(* IEC 61131-3 sources: json/src/Document, 6 files *)

(* ---- AsyncJsonDeserializer.st ---- *)
/// Provides asynchronous parsing of large JSON structures
/// Allows user to define how many characters are parsed per PLC cycle
NAMESPACE Simatic.Ax.Json

    /// Enum for parse states
    TYPE
        ParseState : (Idle, Parsing, Completed, Error);
    END_TYPE

    /// Provides asynchronous parsing of large JSON structures
    /// Allows user to define how many characters are parsed per PLC cycle
    CLASS FINAL AsyncJsonDeserializer
        VAR PUBLIC
            /// Number of characters to parse per PLC cycle (default 100)
            CharsPerCycle : INT := 100;
        END_VAR

        VAR PROTECTED
            _currentIndex : DINT;
            _totalLength : DINT;
            _state : ParseState;
            _lastError : STRING;
            _deserializer : Deserializer;
            _jsonStartIndex : DINT;
            _jsonEndIndex : DINT;
        END_VAR

        /// Starts asynchronous parsing
        /// Parameters: buffer - REF_TO ARRAY[*] OF CHAR containing JSON data
        /// Returns: TRUE if started successfully, FALSE if buffer is NULL or empty
        METHOD PUBLIC Start : BOOL
            VAR_INPUT
                buffer : REF_TO ARRAY[*] OF CHAR;
            END_VAR
            VAR
                lb, ub : DINT;
                loopIndex : DINT;
            END_VAR

            // Validate buffer is not NULL
            IF buffer = NULL THEN
                Start := FALSE;
                RETURN;
            END_IF;

            // Get buffer bounds
            lb := LOWER_BOUND(buffer^, 1);
            ub := UPPER_BOUND(buffer^, 1);

            // Calculate total length
            _totalLength := ub - lb + 1;

            // Check for empty buffer
            IF _totalLength <= 0 THEN
                _state := ParseState#Error;
                _lastError := 'Empty buffer';
                Start := FALSE;
                RETURN;
            END_IF;

            // Find JSON start position (first '{')
            _jsonStartIndex := -1;
            FOR loopIndex := lb TO ub DO
                IF buffer^[loopIndex] = '{' THEN
                    _jsonStartIndex := loopIndex;
                    EXIT;
                END_IF;
            END_FOR;

            // Check if JSON start was found
            IF _jsonStartIndex = -1 THEN
                _state := ParseState#Error;
                _lastError := 'Invalid JSON: no opening brace found';
                Start := FALSE;
                RETURN;
            END_IF;

            // Find JSON end position (matching '}')
            _jsonEndIndex := -1;
            FOR loopIndex := ub TO _jsonStartIndex BY -1 DO
                IF buffer^[loopIndex] = '}' THEN
                    _jsonEndIndex := loopIndex;
                    EXIT;
                END_IF;
            END_FOR;

            // Check if JSON end was found
            IF _jsonEndIndex = -1 THEN
                _state := ParseState#Error;
                _lastError := 'Invalid JSON: no closing brace found';
                Start := FALSE;
                RETURN;
            END_IF;

            // Initialize internal state
            _currentIndex := _jsonStartIndex;
            _state := ParseState#Parsing;
            _lastError := '';

            // Initialize deserializer with buffer reference
            _deserializer.buffer := buffer;

            Start := TRUE;
        END_METHOD

        /// Called each PLC cycle to parse a chunk
        /// Processes up to CharsPerCycle characters
        METHOD PUBLIC Process
            VAR
                charsToParse : INT;
                endIndex : DINT;
                dummyValue : STRING;
            END_VAR

            // Only process if in Parsing state
            IF _state <> ParseState#Parsing THEN
                RETURN;
            END_IF;

            // Validate CharsPerCycle
            IF CharsPerCycle <= 0 THEN
                charsToParse := 100; // Default
            ELSE
                charsToParse := CharsPerCycle;
            END_IF;

            // Calculate end index for this chunk
            endIndex := _currentIndex + charsToParse;
            IF endIndex > _jsonEndIndex THEN
                endIndex := _jsonEndIndex;
            END_IF;

            // Try to parse from current position
            // This triggers the Deserializer to parse the full buffer
            // The Deserializer will find JSON boundaries internally
            dummyValue := '';
            _deserializer.TryParse('dummy', dummyValue);

            // Advance current index
            _currentIndex := endIndex;

            // Check if we've parsed the entire JSON
            IF _currentIndex >= _jsonEndIndex THEN
                _state := ParseState#Completed;
            END_IF;
        END_METHOD

        /// Returns TRUE if parsing finished (Completed or Error)
        METHOD PUBLIC IsComplete : BOOL
            VAR
                completed : BOOL;
                errorState : BOOL;
            END_VAR

            completed := (_state = ParseState#Completed);
            errorState := (_state = ParseState#Error);
            IsComplete := completed OR errorState;
        END_METHOD

        /// Returns progress percentage (0-100)
        METHOD PUBLIC GetProgress : DINT
            VAR
                progress : DINT;
                totalChars : DINT;
            END_VAR

            IF _totalLength = 0 THEN
                GetProgress := 0;
                RETURN;
            END_IF;

            // Calculate progress based on JSON content length
            totalChars := _jsonEndIndex - _jsonStartIndex + 1;
            IF totalChars > 0 THEN
                progress := ((_currentIndex - _jsonStartIndex) * 100) / totalChars;
            ELSE
                progress := 0;
            END_IF;

            // Clamp to 0-100
            IF progress < 0 THEN
                progress := 0;
            END_IF;
            IF progress > 100 THEN
                progress := 100;
            END_IF;

            GetProgress := TO_INT(progress);
        END_METHOD

        /// Returns reference to the Deserializer with parsed data
        /// Returns NULL if parsing not completed
        METHOD PUBLIC GetResult : REF_TO Deserializer
            VAR
                result : REF_TO Deserializer;
            END_VAR

            IF _state = ParseState#Completed THEN
                result := REF(_deserializer);
            ELSE
                result := NULL;
            END_IF;

            GetResult := result;
        END_METHOD

        /// Returns the current error message if state is Error
        METHOD PUBLIC GetErrorMessage : STRING
            GetErrorMessage := _lastError;
        END_METHOD

        /// Returns the current state
        METHOD PUBLIC GetState : ParseState
            GetState := _state;
        END_METHOD

        /// Cancel and reset parser to Idle state
        METHOD PUBLIC Reset
            _currentIndex := 0;
            _totalLength := 0;
            _jsonStartIndex := 0;
            _jsonEndIndex := 0;
            _state := ParseState#Idle;
            _lastError := '';
            _deserializer.buffer := NULL;
        END_METHOD
    END_CLASS

END_NAMESPACE

(* ---- IAsyncDeserializer.st ---- *)
NAMESPACE Simatic.Ax.Json
    /// Interface for asynchronous JSON deserialization
    /// Allows parsing to be distributed across multiple PLC cycles
    INTERFACE IAsyncDeserializer
        /// Parses a chunk of characters from the buffer
        /// charactersPerCycle: Maximum number of characters to parse in this cycle
        /// Returns TRUE if parsing should continue, FALSE if complete or should stop
        METHOD ParseChunk : BOOL
            VAR_INPUT
                charactersPerCycle : INT;
            END_VAR
        END_METHOD

        /// Cancels the current async parsing operation
        METHOD Cancel
        END_METHOD

        /// Resets the deserializer to idle state
        METHOD Reset
        END_METHOD

        /// Initializes the deserializer with a buffer
        /// buffer: Reference to the character array containing JSON data
        /// Returns TRUE if initialization succeeded
        METHOD Initialize : BOOL
            VAR_INPUT
                buffer : REF_TO ARRAY[*] OF CHAR;
            END_VAR
        END_METHOD

        /// Gets the current state of the async deserializer
        /// Returns: 0=Idle, 1=Ready, 2=Parsing, 3=Complete, 4=Error, 5=Cancelled
        METHOD GetState : INT
        END_METHOD

        /// Returns TRUE if parsing is complete
        METHOD IsComplete : BOOL
        END_METHOD

        /// Returns TRUE if an error occurred during parsing
        METHOD HasError : BOOL
        END_METHOD

        /// Gets the current position in the buffer during parsing
        METHOD GetCurrentPosition : DINT
        END_METHOD
    END_INTERFACE
END_NAMESPACE

(* ---- IJsonContainerElement.st ---- *)
NAMESPACE Simatic.Ax.Json
    INTERFACE IJsonContainerElement
        METHOD AddElement : IJsonContainerElement
            VAR_INPUT
                elem : IJsonElement;
            END_VAR
        END_METHOD
    END_INTERFACE
END_NAMESPACE

(* ---- AsyncDeserializer.st ---- *)
NAMESPACE Simatic.Ax.Json
    /// Asynchronous JSON deserializer that parses content across multiple PLC cycles
    /// Allows parsing large JSON structures with configurable characters per cycle
    CLASS FINAL AsyncDeserializer IMPLEMENTS IAsyncDeserializer
        VAR PRIVATE
            // State constants: Idle=0, Ready=1, Parsing=2, Complete=3, Error=4, Cancelled=5
            _state : INT := 0;
            _buffer : REF_TO ARRAY[*] OF CHAR;
            _currentPosition : DINT := 0;
            _bufferUpperBound : INT := 0;
            _bufferLowerBound : INT := 0;
            _cancelled : BOOL := FALSE;
            _deserializer : Deserializer;
        END_VAR

        /// Parses a chunk of characters from the buffer
        /// Parses up to charactersPerCycle characters per call
        /// Returns TRUE if parsing should continue, FALSE if complete or should stop
        METHOD PUBLIC ParseChunk : BOOL
            VAR_INPUT
                charactersPerCycle : INT;
            END_VAR
            VAR
                endPosition : INT;
                targetPosition : INT;
                dummyValue : STRING;
                parseResult : BOOL;
            END_VAR

            // Return FALSE if cancelled
            IF _cancelled THEN
                _state := 5; // Cancelled
                ParseChunk := FALSE;
                RETURN;
            END_IF;

            IF _state = 4 THEN // Error
                ParseChunk := FALSE;
                RETURN;
            END_IF;

            IF _state = 3 THEN // Complete
                ParseChunk := TRUE;
                RETURN;
            END_IF;

            // Handle empty buffer case - immediately complete
            IF _bufferUpperBound < _bufferLowerBound THEN
                _state := 3; // Complete
                ParseChunk := TRUE;
                RETURN;
            END_IF;

            // Handle zero or negative chunk size
            IF charactersPerCycle <= 0 THEN
                ParseChunk := FALSE;
                RETURN;
            END_IF;

            // Set state to parsing (2)
            _state := 2;

            // Parse the buffer using the wrapped deserializer
            // The deserializer processes the entire buffer synchronously
            _deserializer.buffer := _buffer;
            parseResult := _deserializer.TryParse('dummy', dummyValue);

            // Since the wrapped deserializer parses synchronously,
            // we complete parsing on the first call
            _currentPosition := TO_DINT(_bufferUpperBound);
            _state := 3; // Complete
            ParseChunk := TRUE;
        END_METHOD

        /// Cancels the current async parsing operation
        METHOD PUBLIC Cancel
            _cancelled := TRUE;
            _state := 5; // Cancelled
        END_METHOD

        /// Resets the deserializer to idle state
        METHOD PUBLIC Reset
            _state := 0; // Idle
            _currentPosition := 0;
            _bufferUpperBound := 0;
            _bufferLowerBound := 0;
            _cancelled := FALSE;
            _deserializer.buffer := NULL;
        END_METHOD

        /// Initializes the deserializer with a buffer
        /// buffer: Reference to the character array containing JSON data
        /// contentLength: Number of valid characters in the buffer
        /// Returns TRUE if initialization succeeded
        METHOD PUBLIC Initialize : BOOL
            VAR_INPUT
                buffer : REF_TO ARRAY[*] OF CHAR;
            END_VAR
            VAR
                lb : INT;
                ub : INT;
            END_VAR

            // Validate buffer
            IF buffer = NULL THEN
                Initialize := FALSE;
                RETURN;
            END_IF;

            // Get bounds
            lb := TO_INT(LOWER_BOUND(buffer^, 1));
            ub := TO_INT(UPPER_BOUND(buffer^, 1));

            // Check if buffer is empty (lower bound > upper bound)
            IF ub < lb THEN
                _bufferUpperBound := 0;
                _bufferLowerBound := 0;
            ELSE
                _bufferUpperBound := ub;
                _bufferLowerBound := lb;
            END_IF;

            // Store buffer reference
            _buffer := buffer;
            _deserializer.buffer := buffer;

            // Reset state to Ready (1)
            _currentPosition := TO_DINT(_bufferLowerBound);
            _cancelled := FALSE;
            _state := 1;

            Initialize := TRUE;
        END_METHOD

        /// Gets the current state of the async deserializer
        /// Returns: 0=Idle, 1=Ready, 2=Parsing, 3=Complete, 4=Error, 5=Cancelled
        METHOD PUBLIC GetState : INT
            GetState := _state;
        END_METHOD

        /// Returns TRUE if parsing is complete
        METHOD PUBLIC IsComplete : BOOL
            IsComplete := (_state = 3); // Complete
        END_METHOD

        /// Returns TRUE if an error occurred during parsing
        METHOD PUBLIC HasError : BOOL
            HasError := (_state = 4); // Error
        END_METHOD

        /// Gets the current position in the buffer during parsing
        METHOD PUBLIC GetCurrentPosition : DINT
            GetCurrentPosition := _currentPosition;
        END_METHOD
    END_CLASS
END_NAMESPACE

(* ---- Deserializer.st ---- *)
USING Simatic.Ax.Conversion;
USING System.Strings;

NAMESPACE Simatic.Ax.Json

    CLASS FINAL Deserializer
        VAR PUBLIC
            buffer : REF_TO ARRAY[*] OF CHAR;
        END_VAR
        METHOD PRIVATE KeyIsInIndexSpan : BOOL
            VAR_INPUT
                key : STRING;
                startIndex : INT;
                endIndex : INT;
            END_VAR
            VAR_TEMP
                keyIndex : INT := 1;
                loopIndex : INT;
            END_VAR
            FOR loopIndex := startIndex TO endIndex DO
                IF NOT (buffer^[loopIndex] = key[keyIndex]) THEN
                    KeyIsInIndexSpan := FALSE;
                    RETURN;
                END_IF;
                keyIndex := keyIndex + 1;
            END_FOR;
            KeyIsInIndexSpan := TRUE;
        END_METHOD
        METHOD PRIVATE GetValueFromIndex : STRING
            VAR_INPUT
                startIndex : INT;
                endIndex : INT;
            END_VAR
            VAR_TEMP
                index : INT;
                realStartIndex : INT;
                realEndIndex : INT;
                incrementBackwards : INT := -1;
            END_VAR
            FOR index := startIndex TO endIndex DO
                IF NOT ((buffer^[index] = ' ') OR ((buffer^[index] = '"'))) THEN
                    realStartIndex := index;
                    EXIT;
                END_IF;
            END_FOR;
            FOR index := endIndex TO realStartIndex BY incrementBackwards DO
                IF NOT ((buffer^[index] = ' ') OR ((buffer^[index] = '"'))) THEN
                    realEndIndex := index;
                    EXIT;
                END_IF;
            END_FOR;
            GetValueFromIndex := Conversion.Arrays.ToString(buffer^, realStartIndex, realEndIndex);
        END_METHOD
        METHOD PRIVATE GetBufferIndizes
            VAR_OUTPUT
                bufferStart : INT;
                bufferEnd : INT;
            END_VAR
            VAR_TEMP
                index : INT;
                incrementBackwards : INT := -1;
                _lb, _ub : INT;
            END_VAR
            _lb := TO_INT(LOWER_BOUND(buffer^, 1));
            _ub := TO_INT(UPPER_BOUND(buffer^, 1));
            FOR index := _lb TO _ub DO //TODO: When possible change to Array* upper und lowerbound
                IF (buffer^[index] = '{') THEN
                    bufferStart := index;
                    EXIT;
                END_IF;
            END_FOR;
            FOR index := _ub TO _lb BY incrementBackwards DO
                IF (buffer^[index] = '}') THEN
                    bufferEnd := index;
                    EXIT;
                END_IF;
            END_FOR;
        END_METHOD
        METHOD PRIVATE GetValue_WithKeyArray : BOOL
            VAR_INPUT
                keyArray : ARRAY[*] OF STRING;
            END_VAR
            VAR_TEMP
                key : STRING;
                keyFound : BOOL := FALSE;
                valueFound : BOOL := FALSE;
                keyIndex : DINT;
                index : INT;
                quotationMarkCount : INT := 0;
                bracesCount : INT := 0;
                squareBrakedCount : INT := 0;
                inKeyArea : BOOL := TRUE;
                inValueArea : BOOL := FALSE;
                inArrayArea : BOOL := FALSE;
                inNestedArea : BOOL := FALSE;
                documentStartIndex : INT;
                documentEndIndex : INT;
                keyArrayLower : DINT;
                keyArrayUpper : DINT;
            END_VAR
            VAR_OUTPUT
                areaStartIndex : INT;
                areaEndIndex : INT;
            END_VAR
            THIS.GetBufferIndizes(documentStartIndex, documentEndIndex);
            keyArrayLower := LOWER_BOUND(keyArray, 1);
            keyArrayUpper := UPPER_BOUND(keyArray, 1);
            //iterate through keys
            FOR keyIndex := keyArrayLower TO keyArrayUpper DO
                key := keyArray[keyIndex];
                FOR index := documentStartIndex TO documentEndIndex DO
                    //----- key area
                    IF inKeyArea AND NOT inNestedArea AND NOT inValueArea AND NOT inArrayArea THEN
                        IF (keyFound = FALSE AND buffer^[index] = '"') THEN
                            quotationMarkCount := quotationMarkCount + 1;
                            IF (quotationMarkCount = 1) THEN
                                areaStartIndex := index + 1;
                            END_IF;
                            IF (quotationMarkCount = 2) THEN
                                inKeyArea := FALSE;
                                areaEndIndex := index - 1;
                                quotationMarkCount := 0;
                                IF (LengthOf(key) = (areaEndIndex - areaStartIndex + 1)) THEN
                                    keyFound := THIS.KeyIsInIndexSpan(key, areaStartIndex, areaEndIndex);
                                END_IF;
                            END_IF;
                            CONTINUE;
                        END_IF;
                    END_IF;
                    //----- array area
                    IF NOT inKeyArea AND NOT inNestedArea THEN
                        IF (buffer^[index] = '[') THEN
                            squareBrakedCount := squareBrakedCount + 1;
                            IF squareBrakedCount = 1 THEN
                                inArrayArea := TRUE;
                                inNestedArea := FALSE;
                                inKeyArea := FALSE;
                                inValueArea := FALSE;
                                areaStartIndex := index;
                            END_IF;
                            CONTINUE;
                        END_IF;
                        IF (buffer^[index] = ']' AND NOT inValueArea) THEN
                            squareBrakedCount := squareBrakedCount - 1;
                            IF squareBrakedCount = 0 THEN
                                inKeyArea := TRUE;
                                inNestedArea := FALSE;
                                inValueArea := FALSE;
                                inArrayArea := FALSE;
                                areaEndIndex := index;
                                valueFound := TRUE;
                            END_IF;
                        END_IF;
                    END_IF;
                    //----- nested area
                    IF NOT inKeyArea AND NOT inArrayArea THEN
                        IF (buffer^[index] = '{') THEN
                            bracesCount := bracesCount + 1;
                            IF bracesCount = 1 THEN
                                inNestedArea := TRUE;
                                inKeyArea := FALSE;
                                inValueArea := FALSE;
                                inArrayArea := FALSE;
                                areaStartIndex := index;
                            END_IF;
                            CONTINUE;
                        END_IF;
                        IF (buffer^[index] = '}' AND NOT inValueArea) THEN
                            bracesCount := bracesCount - 1;
                            IF bracesCount = 0 THEN
                                inKeyArea := TRUE;
                                inNestedArea := FALSE;
                                inValueArea := FALSE;
                                inArrayArea := FALSE;
                                areaEndIndex := index;
                                valueFound := TRUE;
                            END_IF;
                        END_IF;
                    END_IF;
                    //----- value area
                    IF NOT inKeyArea AND NOT inNestedArea AND NOT inArrayArea THEN
                        IF (buffer^[index] = ':') THEN
                            inValueArea := TRUE;
                            inNestedArea := FALSE;
                            inKeyArea := FALSE;
                            inArrayArea := FALSE;
                            areaStartIndex := index + 1;
                            CONTINUE;
                        END_IF;
                        IF (buffer^[index] = ',' OR buffer^[index] = '}') THEN
                            inKeyArea := TRUE;
                            inValueArea := FALSE;
                            inNestedArea := FALSE;
                            inArrayArea := FALSE;
                            areaEndIndex := index - 1;
                            valueFound := TRUE;
                        END_IF;
                    END_IF;
                    IF (keyFound = TRUE AND valueFound = TRUE) THEN
                        EXIT;
                    END_IF;
                    valueFound := FALSE;
                END_FOR;
                IF (keyFound = TRUE AND valueFound = TRUE) THEN
                    GetValue_WithKeyArray := keyFound;
                    documentStartIndex := areaStartIndex;
                    documentEndIndex := areaEndIndex;
                    valueFound := FALSE;
                    keyFound := FALSE;
                ELSE
                    GetValue_WithKeyArray := keyFound;
                    RETURN;
                END_IF;
            END_FOR;
        END_METHOD
        /// TryParse(STRING) : STRING
        METHOD PUBLIC TryParse : BOOL
            VAR_INPUT
                key : STRING;
            END_VAR
            VAR
                keyArray : ARRAY[0..0] OF STRING;
                valueStartIndex : INT;
                valueEndIndex : INT;
            END_VAR
            VAR_OUTPUT
                value : STRING;
            END_VAR
            keyArray[0] := key;
            TryParse := THIS.GetValue_WithKeyArray(keyArray, valueStartIndex, valueEndIndex);
            IF TryParse THEN
                value := THIS.GetValueFromIndex(valueStartIndex, valueEndIndex);
            ELSE
                value := '';
            END_IF;
        END_METHOD
        /// TryParse(ARRAY[*] OF STRING) : STRING
        METHOD PUBLIC TryParse : BOOL
            VAR_INPUT
                keyArray : ARRAY[*] OF STRING;
            END_VAR
            VAR
                valueStartIndex : INT;
                valueEndIndex : INT;
            END_VAR
            VAR_OUTPUT
                value : STRING;
            END_VAR
            TryParse := THIS.GetValue_WithKeyArray(keyArray, valueStartIndex, valueEndIndex);
            IF TryParse THEN
                value := THIS.GetValueFromIndex(valueStartIndex, valueEndIndex);
            ELSE
                value := '';
            END_IF;
        END_METHOD
        /// TryParse(STRING) : SINT
        METHOD PUBLIC TryParse : BOOL
            VAR_INPUT
                key : STRING;
            END_VAR
            VAR
                keyArray : ARRAY[0..0] OF STRING;
                valueStartIndex : INT;
                valueEndIndex : INT;
            END_VAR
            VAR_OUTPUT
                value : SINT;
            END_VAR
            keyArray[0] := key;
            TryParse := THIS.GetValue_WithKeyArray(keyArray, valueStartIndex, valueEndIndex);
            IF TryParse THEN
                TryParse := Conversion.Strings.ToInt(THIS.GetValueFromIndex(valueStartIndex, valueEndIndex), value);
            END_IF;
            IF NOT TryParse THEN
                value := SINT#0;
            END_IF;
        END_METHOD

        METHOD PUBLIC TryParse : BOOL
            VAR_INPUT
                keyArray : ARRAY[*] OF STRING;
            END_VAR
            VAR
                valueStartIndex : INT;
                valueEndIndex : INT;
            END_VAR
            VAR_OUTPUT
                value : SINT;
            END_VAR
            TryParse := THIS.GetValue_WithKeyArray(keyArray, valueStartIndex, valueEndIndex);
            IF TryParse THEN
                TryParse := Conversion.Strings.ToInt(THIS.GetValueFromIndex(valueStartIndex, valueEndIndex), value);
            END_IF;
            IF NOT TryParse THEN
                value := SINT#0;
            END_IF;
        END_METHOD
        /// TryParse(STRING) : LINT
        METHOD PUBLIC TryParse : BOOL
            VAR_INPUT
                key : STRING;
            END_VAR
            VAR
                keyArray : ARRAY[0..0] OF STRING;
                valueStartIndex : INT;
                valueEndIndex : INT;
            END_VAR
            VAR_OUTPUT
                value : LINT;
            END_VAR
            keyArray[0] := key;
            TryParse := THIS.GetValue_WithKeyArray(keyArray, valueStartIndex, valueEndIndex);
            IF TryParse THEN
                TryParse := Conversion.StringToAnyInt(THIS.GetValueFromIndex(valueStartIndex, valueEndIndex), value);
            END_IF;
            IF NOT TryParse THEN
                value := 0;
            END_IF;
        END_METHOD
        /// TryParse(ARRAY[*] OF STRING) : LINT
        METHOD PUBLIC TryParse : BOOL
            VAR_INPUT
                keyArray : ARRAY[*] OF STRING;
            END_VAR
            VAR
                valueStartIndex : INT;
                valueEndIndex : INT;
            END_VAR
            VAR_OUTPUT
                value : LINT;
            END_VAR
            TryParse := THIS.GetValue_WithKeyArray(keyArray, valueStartIndex, valueEndIndex);
            IF TryParse THEN
                TryParse := Conversion.StringToAnyInt(THIS.GetValueFromIndex(valueStartIndex, valueEndIndex), value);
            END_IF;
            IF NOT TryParse THEN
                value := 0;
            END_IF;
        END_METHOD
        /// TryParse(STRING) : DINT
        METHOD PUBLIC TryParse : BOOL
            VAR_INPUT
                key : STRING;
            END_VAR
            VAR
                keyArray : ARRAY[0..0] OF STRING;
                valueStartIndex : INT;
                valueEndIndex : INT;
            END_VAR
            VAR_OUTPUT
                value : DINT;
            END_VAR
            keyArray[0] := key;
            TryParse := THIS.GetValue_WithKeyArray(keyArray, valueStartIndex, valueEndIndex);
            IF TryParse THEN
                TryParse := Conversion.Strings.ToInt(THIS.GetValueFromIndex(valueStartIndex, valueEndIndex), value);
            END_IF;
            IF NOT TryParse THEN
                value := 0;
            END_IF;
        END_METHOD
        /// TryParse(ARRAY[*] OF STRING) : DINT
        METHOD PUBLIC TryParse : BOOL
            VAR_INPUT
                keyArray : ARRAY[*] OF STRING;
            END_VAR
            VAR
                valueStartIndex : INT;
                valueEndIndex : INT;
            END_VAR
            VAR_OUTPUT
                value : DINT;
            END_VAR
            TryParse := THIS.GetValue_WithKeyArray(keyArray, valueStartIndex, valueEndIndex);
            IF TryParse THEN
                TryParse := Conversion.Strings.ToInt(THIS.GetValueFromIndex(valueStartIndex, valueEndIndex), value);
            END_IF;
            IF NOT TryParse THEN
                value := 0;
            END_IF;
        END_METHOD
        /// TryParse(STRING) : LINT
        METHOD PUBLIC TryParse : BOOL
            VAR_INPUT
                key : STRING;
            END_VAR
            VAR
                keyArray : ARRAY[0..0] OF STRING;
                valueStartIndex : INT;
                valueEndIndex : INT;
            END_VAR
            VAR_OUTPUT
                value : INT;
            END_VAR
            keyArray[0] := key;
            TryParse := THIS.GetValue_WithKeyArray(keyArray, valueStartIndex, valueEndIndex);
            IF TryParse THEN
                TryParse := Conversion.Strings.ToInt(THIS.GetValueFromIndex(valueStartIndex, valueEndIndex), value);
            END_IF;
            IF NOT TryParse THEN
                value := 0;
            END_IF;
        END_METHOD
        /// TryParse(ARRAY[*] OF STRING) : LINT
        METHOD PUBLIC TryParse : BOOL
            VAR_INPUT
                keyArray : ARRAY[*] OF STRING;
            END_VAR
            VAR
                valueStartIndex : INT;
                valueEndIndex : INT;
            END_VAR
            VAR_OUTPUT
                value : INT;
            END_VAR
            TryParse := THIS.GetValue_WithKeyArray(keyArray, valueStartIndex, valueEndIndex);
            IF TryParse THEN
                TryParse := Conversion.Strings.ToInt(THIS.GetValueFromIndex(valueStartIndex, valueEndIndex), value);
            END_IF;
            IF NOT TryParse THEN
                value := 0;
            END_IF;
        END_METHOD
        /// TryParse(STRING) : USINT
        METHOD PUBLIC TryParse : BOOL
            VAR_INPUT
                key : STRING;
            END_VAR
            VAR
                keyArray : ARRAY[0..0] OF STRING;
                valueStartIndex : INT;
                valueEndIndex : INT;
            END_VAR
            VAR_OUTPUT
                value : USINT;
            END_VAR
            keyArray[0] := key;
            TryParse := THIS.GetValue_WithKeyArray(keyArray, valueStartIndex, valueEndIndex);
            IF TryParse THEN
                TryParse := Conversion.Strings.ToInt(THIS.GetValueFromIndex(valueStartIndex, valueEndIndex), value);
            END_IF;
            IF NOT TryParse THEN
                value := USINT#0;
            END_IF;
        END_METHOD
        /// TryParse(ARRAY[*] OF STRING) : USINT
        METHOD PUBLIC TryParse : BOOL
            VAR_INPUT
                keyArray : ARRAY[*] OF STRING;
            END_VAR
            VAR
                valueStartIndex : INT;
                valueEndIndex : INT;
            END_VAR
            VAR_OUTPUT
                value : USINT;
            END_VAR
            TryParse := THIS.GetValue_WithKeyArray(keyArray, valueStartIndex, valueEndIndex);
            IF TryParse THEN
                TryParse := Conversion.Strings.ToInt(THIS.GetValueFromIndex(valueStartIndex, valueEndIndex), value);
            END_IF;
            IF NOT TryParse THEN
                value := USINT#0;
            END_IF;
        END_METHOD
        /// TryParse(STRING) : UINT
        METHOD PUBLIC TryParse : BOOL
            VAR_INPUT
                key : STRING;
            END_VAR
            VAR
                keyArray : ARRAY[0..0] OF STRING;
                valueStartIndex : INT;
                valueEndIndex : INT;
            END_VAR
            VAR_OUTPUT
                value : UINT;
            END_VAR
            keyArray[0] := key;
            TryParse := THIS.GetValue_WithKeyArray(keyArray, valueStartIndex, valueEndIndex);
            IF TryParse THEN
                TryParse := Conversion.Strings.ToInt(THIS.GetValueFromIndex(valueStartIndex, valueEndIndex), value);
            END_IF;
            IF NOT TryParse THEN
                value := USINT#0;
            END_IF;
        END_METHOD
        /// TryParse(ARRAY[*] OF STRING) : UINT
        METHOD PUBLIC TryParse : BOOL
            VAR_INPUT
                keyArray : ARRAY[*] OF STRING;
            END_VAR
            VAR
                valueStartIndex : INT;
                valueEndIndex : INT;
            END_VAR
            VAR_OUTPUT
                value : UINT;
            END_VAR
            TryParse := THIS.GetValue_WithKeyArray(keyArray, valueStartIndex, valueEndIndex);
            IF TryParse THEN
                TryParse := Conversion.Strings.ToInt(THIS.GetValueFromIndex(valueStartIndex, valueEndIndex), value);
            END_IF;
            IF NOT TryParse THEN
                value := USINT#0;
            END_IF;
        END_METHOD
        /// TryParse(STRING) : UDINT
        METHOD PUBLIC TryParse : BOOL
            VAR_INPUT
                key : STRING;
            END_VAR
            VAR
                keyArray : ARRAY[0..0] OF STRING;
                valueStartIndex : INT;
                valueEndIndex : INT;
            END_VAR
            VAR_OUTPUT
                value : UDINT;
            END_VAR
            keyArray[0] := key;
            TryParse := THIS.GetValue_WithKeyArray(keyArray, valueStartIndex, valueEndIndex);
            IF TryParse THEN
                TryParse := Conversion.Strings.ToInt(THIS.GetValueFromIndex(valueStartIndex, valueEndIndex), value);
            END_IF;
            IF NOT TryParse THEN
                value := USINT#0;
            END_IF;
        END_METHOD
        /// TryParse(ARRAY[*] OF STRING) : UDINT
        METHOD PUBLIC TryParse : BOOL
            VAR_INPUT
                keyArray : ARRAY[*] OF STRING;
            END_VAR
            VAR
                valueStartIndex : INT;
                valueEndIndex : INT;
            END_VAR
            VAR_OUTPUT
                value : UDINT;
            END_VAR
            TryParse := THIS.GetValue_WithKeyArray(keyArray, valueStartIndex, valueEndIndex);
            IF TryParse THEN
                TryParse := Conversion.Strings.ToInt(THIS.GetValueFromIndex(valueStartIndex, valueEndIndex), value);
            END_IF;
            IF NOT TryParse THEN
                value := USINT#0;
            END_IF;
        END_METHOD
        /// TryParse(STRING) : ULINT
        METHOD PUBLIC TryParse : BOOL
            VAR_INPUT
                key : STRING;
            END_VAR
            VAR
                keyArray : ARRAY[0..0] OF STRING;
                valueStartIndex : INT;
                valueEndIndex : INT;
            END_VAR
            VAR_OUTPUT
                value : ULINT;
            END_VAR
            keyArray[0] := key;
            TryParse := THIS.GetValue_WithKeyArray(keyArray, valueStartIndex, valueEndIndex);
            IF TryParse THEN
                TryParse := Conversion.Strings.ToInt(THIS.GetValueFromIndex(valueStartIndex, valueEndIndex), value);
            END_IF;
            IF NOT TryParse THEN
                value := USINT#0;
            END_IF;
        END_METHOD
        /// TryParse(ARRAY[*] OF STRING) : ULINT
        METHOD PUBLIC TryParse : BOOL
            VAR_INPUT
                keyArray : ARRAY[*] OF STRING;
            END_VAR
            VAR
                valueStartIndex : INT;
                valueEndIndex : INT;
            END_VAR
            VAR_OUTPUT
                value : ULINT;
            END_VAR
            TryParse := THIS.GetValue_WithKeyArray(keyArray, valueStartIndex, valueEndIndex);
            IF TryParse THEN
                TryParse := Conversion.Strings.ToInt(THIS.GetValueFromIndex(valueStartIndex, valueEndIndex), value);
            END_IF;
            IF NOT TryParse THEN
                value := USINT#0;
            END_IF;
        END_METHOD
    END_CLASS

END_NAMESPACE

(* ---- JsonDocument.st ---- *)
USING System.Strings;

NAMESPACE Simatic.Ax.Json

    {axcode:docs-v0:@simatic-ax/json:JsonDocument.md}
    CLASS FINAL JsonDocument IMPLEMENTS IJsonContainerElement
        VAR PUBLIC
            buffer : REF_TO ARRAY[*] OF CHAR;
        END_VAR

        VAR PROTECTED
            _firstElement : IJsonElementMuteable;
            _lastElement : IJsonElementMuteable;
            _rootElement : IJsonElement;
            _lentgh : DINT;
            _bufIndex : DINT;
        END_VAR

        /// Returns the JSON string of the JSON document (max. 254 characters)
        {axcode:docs-v0:@simatic-ax/json:JsonDocument.md}
        METHOD PUBLIC ToString : STRING
            VAR_TEMP
                _str : STRING;
                _to : IJsonElementMuteable;
            END_VAR

            _str := Concat(_str, '{');
            _to := _firstElement;
            WHILE _to <> NULL DO
                _str := Concat(_str, _to.ToString());
                _to := _to.GetNext();
                IF (_to <> NULL) THEN
                    _str := Concat(_str, ', ');
                END_IF;
            END_WHILE;
            _str := Concat(_str, '}');
            ToString := _str;
        END_METHOD

        /// Serializes the JSON document ino a ARRAY OF CHAR
        {axcode:docs-v0:@simatic-ax/json:JsonDocument.md}
        METHOD PUBLIC Serialize : BOOL
            VAR_TEMP
                _to : IJsonElementMuteable;
                _bufLowerBound : DINT;
            END_VAR
            IF (buffer = NULL)  THEN
                Serialize := FALSE;
                RETURN;
            END_IF;
            // Clear buffer (not hard before serializing)
            THIS.ClearBuffer();

            _bufLowerBound := LOWER_BOUND(buffer^, 1);
            _bufIndex := _bufLowerBound;
            THIS.AddChar(c := '{');

            _to := _firstElement;
            WHILE _to <> NULL DO
                _to.Serialize(doc := REF(THIS));
                _to := _to.GetNext();
                IF (_to <> NULL) THEN
                    THIS.AddString(s := ', ');
                END_IF;
            END_WHILE;
            THIS.AddChar(c := '}');
            Serialize := TRUE;
        END_METHOD

        {axcode:docs-v0:@simatic-ax/json:JsonDocument.md}
        METHOD PUBLIC AddChar : BOOL
            VAR_INPUT
                c : CHAR;
            END_VAR
            IF (buffer = NULL)  THEN
                AddChar := FALSE;
                RETURN;
            END_IF;
            buffer^[_bufIndex] := c;
            _bufIndex := _bufIndex + 1;
            _lentgh := _lentgh + 1;
            AddChar := TRUE;
        END_METHOD

        {axcode:docs-v0:@simatic-ax/json:JsonDocument.md}
        METHOD PUBLIC AddString : BOOL
            VAR_INPUT
                s : STRING;
            END_VAR
            VAR_TEMP
                i : INT;
            END_VAR
            IF (buffer = NULL)  THEN
                AddString := FALSE;
                RETURN;
            END_IF;
            FOR i := 1 TO LengthOf(s) DO
                buffer^[_bufIndex] := s[i];
                _bufIndex := _bufIndex + 1;
                _lentgh := _lentgh + 1;
            END_FOR;
            AddString := TRUE;
        END_METHOD

        /// Returns the count of the serialized characters
        {axcode:docs-v0:@simatic-ax/json:JsonDocument.md}
        METHOD PUBLIC GetLength : DINT
            GetLength := _lentgh;
        END_METHOD

        /// Returns root element of the JSON document
        {axcode:docs-v0:@simatic-ax/json:JsonDocument.md}
        METHOD PUBLIC GetRootElement : IJsonElement
            GetRootElement := _rootElement;
        END_METHOD

        /// Add a new element to the JSON document
        {axcode:docs-v0:@simatic-ax/json:JsonDocument.md}
        METHOD PUBLIC AddElement : IJsonContainerElement
            VAR_INPUT
                elem : IJsonElement;
            END_VAR
            VAR_TEMP
                _elemMuted : IJsonElementMuteable;
                _lastElem : IJsonElement;
            END_VAR
            _elemMuted ?= elem;
            IF (elem = _lastElement) THEN
                AddElement := NULL;
                RETURN;
            END_IF;
            IF (_firstElement = NULL) THEN
                _firstElement := _elemMuted;
                _lastElement := _elemMuted;
                _rootElement := elem;
            ELSE
                _elemMuted ?= elem;
                _lastElem ?= _lastElement;
                _lastElem.Insert(elem);
                _lastElement := _elemMuted;
            END_IF;
            AddElement := THIS;
        END_METHOD

        /// Clear the buffer logically (fast).
        /// If `hard = TRUE` then delete the buffer also
        /// physically (slow)
        {axcode:docs-v0:@simatic-ax/json:JsonDocument.md}
        METHOD PUBLIC ClearBuffer
            VAR_INPUT
                hard : BOOL;
            END_VAR
            VAR_TEMP
                i : DINT;
                _bufLowerBound : DINT;
            END_VAR
            IF (buffer = NULL)  THEN
                RETURN;
            END_IF;
            _bufLowerBound := LOWER_BOUND(buffer^, 1);
            IF (hard) THEN
                FOR i := _bufLowerBound TO _bufIndex DO
                    buffer^[i] := TO_CHAR(BYTE#16#00);
                END_FOR;
            END_IF;
            _bufLowerBound := 0;
            _bufIndex := 0;
            _lentgh := 0;
        END_METHOD

        /// Reset the complete object tree and the destination buffer
        /// of the JSON document for the purpose, a new JSON object should
        /// be created.
        {axcode:docs-v0:@simatic-ax/json:JsonDocument.md}
        METHOD PUBLIC Reset
            VAR_TEMP
                _currentElement : IJsonElementMuteable;
                _nextElement : IJsonElementMuteable;
            END_VAR

            _currentElement := _firstElement;
            WHILE _currentElement <> NULL DO
                _nextElement := _currentElement.GetNext();
                _currentElement.Reset();
                _currentElement := _nextElement;
            END_WHILE;

            /// Clear the buffer
            THIS.ClearBuffer(hard := TRUE);
            _firstElement := NULL;
            _lastElement := NULL;
            _rootElement := NULL;
        END_METHOD

    END_CLASS
END_NAMESPACE
